TYPE ForceMeasurementStatuses :
STRUCT
	///Is the force being measured?
	enabledStatus: EnabledStatus;
	///Is the measurement OK?
	healthStatus: HealthStatus;
	///Alarm status
	alarmStatus: HiHiLoLoAlarmStatus;
END_STRUCT
END_TYPE

(* stored: Version 1.1.0.1, ProductVersion 3.1.4019.2
   DUT ForceMeasurementStatuses: Id {f6795bfb-a451-4af6-be54-859153c1f796} *)
